FUNCTION_BLOCK FB_StateLogger IMPLEMENTS I_Logger
VAR
END_VAR

METHOD M_Log
VAR_INPUT
	stEvent	: 		ST_Event;
END_VAR
END_METHOD

END_FUNCTION_BLOCK

(* stored: Version 1.1.0.1
   POU FB_StateLogger: Id {f96c5de2-5f35-067d-1150-42c81efb44d8}, SpecialFunc None
   Method M_Log: Id {f2b4e8fe-9036-054e-2b03-2a61e7ff6ae3} *)
